(* IEC 61131-3 sources: AXOpen/src/templates.simple/ax/src/templates/starterunit, 8 files *)

(* ---- AutomatSequence.st ---- *)
NAMESPACE axosimple.StarterUnitTemplate
    USING axosimple;
    USING AXOpen.Data;
    USING AXOpen.Core;
    USING System.Strings;

    ///<summary>
    /// Provides automatic mode sequence.
    ///</summary>
    {#ix-set:AttributeName = "<#AUTOMAT#>"}
    {S7.extern=ReadWrite}
    CLASS PUBLIC AutomatSequence
        EXTENDS AXOpen.Core.AxoSequencerContainer IMPLEMENTS IModeContainer
        VAR PUBLIC
            Steps : ARRAY[0..100] OF AxoStep;

            _inspectionResult: BOOL;
            _inspectionValue: LREAL;
            _inspectionData: STRING;

            _comprehensiveResult: AXOpen.Inspectors.AxoComprehensiveResult;
        END_VAR

        VAR PRIVATE
            Objs : REF_TO axosimple.StarterUnitTemplate.UnitObjects;
            Components : REF_TO axosimple.StarterUnitTemplate.Components;
            ProcessDataManager : REF_TO axosimple.StarterUnitTemplate.ProcessDataManager;
            ProcessSettingsManager : REF_TO axosimple.StarterUnitTemplate.FragmentProcessDataManger;
            TechnologySettingsManager : REF_TO axosimple.StarterUnitTemplate.TechnologyDataManager;

            EntityHeader : REF_TO axosimple.EntityData;
            ProcessData : REF_TO axosimple.StarterUnitTemplate.ProcessData;
            ProcessSettings : REF_TO axosimple.StarterUnitTemplate.ProcessData;
            TechnologySettings : REF_TO axosimple.StarterUnitTemplate.TechnologyData;

            _currentId : STRING;

            _dialogAnswer : eDialogAnswer;
            _externalCloseOkSignal : BOOL;
        END_VAR

        METHOD INTERNAL Run
            VAR_INPUT
                _parent : AXOpen.Core.IAxoObject;
                _unitObjects : REF_TO UnitObjects;
            END_VAR

            IF Objs = NULL THEN
                Objs := _unitObjects;

                Components := Objs^.Components;
                ProcessDataManager := Objs^.ProcessData;
                ProcessSettingsManager := Objs^.ProcessSettings;
                TechnologySettingsManager := Objs^.TechnologySettings;

                EntityHeader := REF(ProcessDataManager^.Shared.Entity);
                ProcessData :=  REF(ProcessDataManager^.DataManger.Payload);
                ProcessSettings :=  REF(ProcessSettingsManager^.Payload);
                TechnologySettings :=  REF(TechnologySettingsManager^.DataManger.Payload);

            END_IF;

            SUPER.Run(_parent);
        END_METHOD
        ///<summary>
        /// Contains logic of the steps of this sequence
        ///</summary>

        METHOD OVERRIDE Main
            VAR
                forIterator : INT := 0;
                dialogTimeOut : TIME:= t#3000ms;
            END_VAR

            IF (Components = NULL OR ProcessDataManager = NULL) THEN
                RETURN;
            END_IF;
            // This sequecner executes the steps in cycles from top to bottom
            // in the same order they are written in the program
            // Each step in the sequence must can be used only once.
            // This sets the sequence to run in cycles (top-botton-top and again).
            THIS.SequenceMode := eAxoSequenceMode#Cyclic;

            IF (Steps[0].Execute(THIS, TRUE, '<#GET ID#>')) THEN
                //-------------------------------------------------------
                Objs^._inspectorDialog.Restore();

                // copy data from setting to station data -> it's a problem with override checks identity
                //ProcessData^ :=  ProcessSettings^;

                ProcessData^.PartPresence.Data()^.FailTime := TIME#3s;
                ProcessData^.LoadPosition.Data()^.FailTime := TIME#3s;
                ProcessData^.JigDataMatrixCode.Data()^.FailTime := TIME#3s;

                ProcessData^.PartPresence.Data()^.PassTime := TIME#2.5s;
                ProcessData^.LoadPosition.Data()^.PassTime := TIME#2s;
                ProcessData^.JigDataMatrixCode.Data()^.PassTime := TIME#2s;

                ProcessData^.PartPresence.Data()^.RequiredStatus := TRUE;
                ProcessData^.LoadPosition.Data()^.RequiredMin := 1000.0;
                ProcessData^.LoadPosition.Data()^.RequiredMax := 2000.0;
                ProcessData^.JigDataMatrixCode.Data()^.RequiredStatus := 'passCode';

                _currentId := 'newProducedPart';
                THIS.MoveNext();
                //-------------------------------------------------------
            END_IF;

            IF (Steps[1].Execute(THIS, TRUE, '<#GET DATA#>')) THEN
                //-------------------------------------------------------
                IF (ProcessDataManager^.CreateOrUpdate(_currentId).IsDone()) THEN
                    THIS.MoveNext();
                END_IF;
                //-------------------------------------------------------
            END_IF;

            IF (Steps[2].Execute(THIS, TRUE, '<#Dialog notify#>')) THEN
                //-------------------------------------------------------
                _externalCloseOkSignal := CurrentStep.Duration > dialogTimeOut;

                _dialogAnswer := Objs^._dialog.ShowWithExternalClose(THIS, _externalCloseOkSignal)
                .WithOK()
                .WithType(eDialogType#Info)
                .WithCaption('Info caption!')
                .WithText('Info - dialog will be closed by external timeout 2s!').Answer();

                IF( _dialogAnswer = eDialogAnswer#Ok) THEN
                    THIS.MoveNext();
                END_IF;
                //-------------------------------------------------------
            END_IF;

            IF (Steps[3].Execute(THIS, TRUE, '<#Dialog success#>')) THEN
                //-------------------------------------------------------
                _externalCloseOkSignal := CurrentStep.Duration > dialogTimeOut;

                    _dialogAnswer := Objs^._dialog.ShowWithExternalClose(THIS, _externalCloseOkSignal)
                    .WithOK()
                    .WithType(eDialogType#Success)
                    .WithCaption('Success caption!')
                    .WithText('Success - dialog will be closed by external timeout 2s!').Answer();

                    IF( _dialogAnswer = eDialogAnswer#Ok) THEN
                        THIS.MoveNext();
                    END_IF;
                //-------------------------------------------------------
            END_IF;

            IF (Steps[4].Execute(THIS, TRUE, '<#Dialog Warning#>')) THEN
                //-------------------------------------------------------
                _externalCloseOkSignal := CurrentStep.Duration > dialogTimeOut;

                    _dialogAnswer := Objs^._dialog.ShowWithExternalClose(THIS, _externalCloseOkSignal)
                    .WithYesNo()
                    .WithType(eDialogType#Warning)
                    .WithCaption('Warning caption!')
                    .WithText('Warning - dialog will be closed by external timeout 2s!').Answer();

                    IF( _dialogAnswer = eDialogAnswer#Ok) THEN
                        THIS.MoveNext();
                    END_IF;
                //-------------------------------------------------------
            END_IF;

            IF (Steps[5].Execute(THIS, TRUE, '<#Dialog danger#>')) THEN
                //-------------------------------------------------------
                _externalCloseOkSignal := CurrentStep.Duration > dialogTimeOut;

                    _dialogAnswer := Objs^._dialog.ShowWithExternalClose(THIS, _externalCloseOkSignal)
                    .WithYesNoCancel()
                    .WithType(eDialogType#Warning)
                    .WithCaption('Danger caption!')
                    .WithText('Danger - dialog will be closed by external timeout 2s!').Answer();

                    IF( _dialogAnswer = eDialogAnswer#Ok) THEN
                        THIS.MoveNext();
                    END_IF;
                //-------------------------------------------------------
            END_IF;

            IF (Steps[6].Execute(THIS, TRUE, 'Example Digital inspection')) THEN
                //-------------------------------------------------------
                ProcessData^.PartPresence.WithCoordinator(THIS).Inspect(THIS,_inspectionResult)
                .UpdateComprehensiveResult(_comprehensiveResult)
                .OnFail()
                .CarryOn();
                //-------------------------------------------------------
            END_IF;

            IF (Steps[7].Execute(THIS, TRUE, 'Example Analog inspection')) THEN
                //-------------------------------------------------------
                _inspectionValue := -5500;

                ProcessData^.LoadPosition.WithCoordinator(THIS)
                .Inspect(THIS,_inspectionValue)
                .UpdateComprehensiveResult(_comprehensiveResult)
                .OnFail()
                .Dialog( inRetryStep := Steps[50], inTerminateStep := Steps[60], inoDialog := Objs^._inspectorDialog);
                //-------------------------------------------------------
            END_IF;

            IF (Steps[8].Execute(THIS, TRUE, 'Example Data inspection')) THEN
                //-------------------------------------------------------
                _inspectionData := 'tempCode';

                ProcessData^.JigDataMatrixCode.WithCoordinator(THIS)
                .Inspect(THIS,_inspectionData)
                .UpdateComprehensiveResult(_comprehensiveResult)
                .OnFail()
                .Dialog( inRetryStep := Steps[70], inTerminateStep := Steps[80], inoDialog := Objs^._inspectorDialog);
                //-------------------------------------------------------
            END_IF;

            FOR forIterator := 10 TO 89 BY 1 DO
                IF (Steps[forIterator].Execute(THIS, TRUE,Concat('DO SOMETHING -A-',ToString(forIterator)) )) THEN
                    //-------------------------------------------------------
                    IF CurrentStep.Duration > TIME#50ms THEN
                        THIS.MoveNext();
                    END_IF;
                    //-------------------------------------------------------
                END_IF;
            END_FOR;

            IF (Steps[99].Execute(THIS, TRUE,'<#UPDATE DATA#>')) THEN
                //-------------------------------------------------------
                IF (ProcessDataManager^.Update(_currentId).IsDone()) THEN
                    THIS.MoveNext();
                END_IF;
                //-------------------------------------------------------
            END_IF;

            // This will close the sequence and will return to the first step.
            THIS.Close(Steps[100]);
        END_METHOD
    END_CLASS

END_NAMESPACE

(* ---- Comonents.st ---- *)
NAMESPACE axosimple.StarterUnitTemplate
    USING axosimple;
    USING AXOpen.Data;
    USING AXOpen.Core;
    USING System.Strings;

    ///<summary>
    /// Groups components of this controller unit.
    ///</summary>
    {S7.extern=ReadWrite}
    CLASS Components
        EXTENDS AXOpen.Core.AxoObject
        VAR PUBLIC
            // HERE DECLARE COMPONENTS USED BY THIS CONTROLLED UNIT
            // HorizontalCylinder : AXOpen.Components.Pneumatics.AxoCylinder;
            // VerticalCylinder : AXOpen.Components.Pneumatics.AxoCylinder;
            // GripperCylinder : AXOpen.Components.Pneumatics.AxoCylinder;
            // DMCReader : AXOpen.Components.Cognex.Vision.v_6_0_0_0.AxoDataman;
            // PartPresenceSensor : AXOpen.Elements.AxoDi;
        END_VAR

        METHOD PUBLIC Update
            VAR_INPUT
                parent : IAxoObject;
            END_VAR
            VAR_IN_OUT
                Inputs : axosimple.Inputs;
                Outputs : axosimple.Outputs;
            END_VAR
            THIS.Initialize(parent);
            // HERE INITIALIZE YOUR COMPONENTS
            // HorizontalCylinder.Run(THIS, Inputs.B0[0], Inputs.B0[1], Outputs.B0[0], Outputs.B0[1]);
            // VerticalCylinder.Run(THIS, Inputs.B0[2], Inputs.B0[3], Outputs.B0[2], Outputs.B0[3]);
            // GripperCylinder.Run(THIS, Inputs.B0[4], Inputs.B0[5], Outputs.B0[4], Outputs.B0[5]);
        END_METHOD
    END_CLASS
END_NAMESPACE

(* ---- GroundSequence.st ---- *)
NAMESPACE axosimple.StarterUnitTemplate
    USING axosimple;
    USING AXOpen.Data;
    USING AXOpen.Core;
    USING System.Strings;

    ///<summary>
    /// Provides ground mode sequence.
    ///</summary>
    {#ix-set:AttributeName = "<#GROUND#>"}
    {S7.extern=ReadWrite}
    CLASS PUBLIC GroundSequence
        EXTENDS AXOpen.Core.AxoSequencerContainer
        VAR PUBLIC
            Steps : ARRAY[0..20] OF AxoStep;
            MoveToWork : AxoTask;
        END_VAR
        VAR PRIVATE
            Objs : REF_TO axosimple.StarterUnitTemplate.UnitObjects;
            Components : REF_TO Components;
            ProcessData : REF_TO ProcessDataManager;
            ProcessSettings : REF_TO FragmentProcessDataManger;
            TechnologySettings : REF_TO TechnologyDataManager;
            PersistentSettings : REF_TO AxoDataPersistentExchange;

            _currentId : STRING;
            techSetttingsId : STRING;
        END_VAR

        METHOD INTERNAL Run
            VAR_INPUT
                _parent : IAxoObject;
                _unitObjects : REF_TO axosimple.StarterUnitTemplate.UnitObjects;
            END_VAR

            IF Objs = NULL THEN
                Objs := _unitObjects;

                Components := Ref(Objs^.Components);
                ProcessData := Objs^.ProcessData;
                ProcessSettings := Objs^.ProcessSettings;
                TechnologySettings := Objs^.TechnologySettings;
                PersistentSettings := Objs^.Global^.PersistentData;
            END_IF;

            SUPER.Run(_parent);
        END_METHOD

        ///<summary>
        /// Contains logic of the steps of this sequence
        ///</summary>
        METHOD PROTECTED OVERRIDE Main
            VAR
                taskState :IAxoTaskState;
            END_VAR;
            // IF (Components = NULL OR ProcessData = NULL) THEN
            //     RETURN;
            // END_IF;
            // This sequecner executes the steps in cycles from top to bottom
            // in the same order they are written in the program
            // Each step in the sequence must can be used only once.
            // This sets the sequence to run once (top-botton) and stops with done after closing.
            THIS.SequenceMode := eAxoSequenceMode#RunOnce;

            // This is more verbose but also more versatile way of executing step logic.
            IF (Steps[0].Execute(THIS, TRUE, '<#RESTORE#>')) THEN
                //-------------------------------------------------------
                TechnologySettings^.Restore();
                ProcessSettings^.Restore();
                ProcessData^.Restore();

                THIS.MoveNext();
                //-------------------------------------------------------
            END_IF;

            IF (Steps[1].Execute(THIS, TRUE, '<#READ PERSISTENT SETTINGS#>')) THEN
                //-------------------------------------------------------
                IF CurrentStep.IsFirstEntryToStep() THEN
                    ;// some special initialization
                END_IF;

                CASE TO_INT( THIS.GetMicroStepValue()) OF
                    0 :
                        IF PersistentSettings^.InvokeEntityExist(THIS ,'') THEN
                            THIS.SetMicroStepValue(UINT#10);
                        END_IF;

                    10 :
                        IF PersistentSettings^.IsEntityExistDone(THIS) THEN
                            IF PersistentSettings^.EntityExistResult() THEN
                                THIS.SetMicroStepValue(UINT#40); // default data exist
                            ELSE
                                THIS.SetMicroStepValue(UINT#20); // no data exist
                            END_IF;
                        END_IF;

                    20 :
                        IF PersistentSettings^.InvokeUpdateAll(THIS) THEN // data not exist -> udate all to DB
                            THIS.SetMicroStepValue(UINT#30);
                        END_IF;

                    30:
                        IF PersistentSettings^.IsUpdateAllDone(THIS) THEN
                            THIS.SetMicroStepValue(UINT#40); // all was updated to DB
                        END_IF;

                    40 :
                        IF PersistentSettings^.InvokeRead(THIS, '') THEN // read default group
                            THIS.SetMicroStepValue(UINT#50);
                        END_IF;
                    50 :
                        IF PersistentSettings^.IsReadDone(THIS) THEN
                                THIS.MoveNext(); // just default group was readed
                        END_IF;
                    ELSE
                        THIS.SetMicroStepValue(UINT#0);
                END_CASE;

                //-------------------------------------------------------
            END_IF;

            IF (Steps[5].Execute(THIS, TRUE, '<#READ TECHNOLOGY SETTINS#>')) THEN
                //-------------------------------------------------------
                IF CurrentStep.IsFirstEntryToStep() THEN

                    IF Objs^.Global^.TechnologySettings^.Common.Entity.DataEntityId <> '' THEN
                       techSetttingsId := Objs^.Global^.TechnologySettings^.Common.Entity.DataEntityId; // TAKE GLOGAL TECHNOLOGY SETTINGS ID

                    ELSIF Objs^.TechnologySettings^.Shared.Entity.DataEntityId <> '' THEN // TAKE LAST LOADED FOR STATION
                        techSetttingsId := Objs^.TechnologySettings^.Shared.Entity.DataEntityId;

                    ELSIF Objs^.LastTechnologySettings <> '' THEN // TAKE LAST LOADED FROM PERSISTENT
                        techSetttingsId := Objs^.LastTechnologySettings;
                    ELSE
                        Objs^.LastTechnologySettings := 'default'; // FORCE DEFAULT VALUE
                        techSetttingsId := Objs^.LastTechnologySettings;
                    END_IF;

                    IF Objs^.Global^.TechnologySettings^.Common.Entity.DataEntityId = Objs^.TechnologySettings^.Shared.Entity.DataEntityId then
                        //THIS.MoveNext(); // you can skip loading...
                        ;
                    end_if;

                else
                    IF(TechnologySettings^.Read( techSetttingsId ).IsDone()) THEN
                        THIS.MoveNext();
                    END_IF;
                END_IF;
                //-------------------------------------------------------
            END_IF;

            IF (Steps[6].Execute(THIS, TRUE, '<#DO SOMETHING#>')) THEN
                //-------------------------------------------------------
                IF CurrentStep.Duration > TIME#2s THEN
                    THIS.MoveNext();
                END_IF;
                //-------------------------------------------------------
            END_IF;

            IF (Steps[19].Execute(THIS, TRUE, '<#SAVE DATA#>')) THEN
                //-------------------------------------------------------
                CASE TO_INT( THIS.GetMicroStepValue()) OF
                    0 :
                        IF ProcessData^.Shared.Entity.DataEntityId <> '' THEN
                            _currentId := ProcessData^.Shared.Entity.DataEntityId;
                            THIS.SetMicroStepValue(UINT#10);

                        ELSE // FIST RUN OR WITHOUT DATA
                            THIS.MoveNext();
                        END_IF;

                    10 : // update part as a corrupted a interrupted
                        ProcessData^.Shared.Entity.WasReset := true;
                        IF ProcessData^.Update(_currentId).IsDone() THEN
                                THIS.MoveNext();
                        END_IF;
                    ELSE
                        THIS.SetMicroStepValue(UINT#0);
                END_CASE;
                //-------------------------------------------------------
            END_IF;

            // This will close the sequence and will return to the first step.
            THIS.Close(Steps[20]);
        END_METHOD
    END_CLASS
END_NAMESPACE

(* ---- ProcessData.st ---- *)
NAMESPACE axosimple.StarterUnitTemplate
    USING axosimple;
    USING AXOpen.Data;
    USING AXOpen.Core;
    USING System.Strings;

    {S7.extern=ReadWrite}
    CLASS ProcessData
        EXTENDS AXOpen.Data.AxoDataEntity
        VAR PUBLIC
            CounterDelay : ULINT;
        END_VAR
    END_CLASS
END_NAMESPACE

(* ---- ServiceMode.st ---- *)
NAMESPACE axosimple.StarterUnitTemplate
    USING axosimple;
    USING AXOpen.Data;
    USING AXOpen.Core;
    USING System.Strings;

    ///<summary>
    /// Provides logic for service/manual/maintenance mode.
    ///</summary>
    {#ix-set:AttributeName = "<#SERVICE#>"}
    {S7.extern=ReadWrite}
    CLASS PUBLIC ServiceMode
        EXTENDS AXOpen.Core.AxoTask
        ///<summary>
        /// Runs service mode logic. This method must be called cyclically.
        ///</summary>

        METHOD PUBLIC Run
            VAR_INPUT
                parent : IAxoObject;
            END_VAR
            VAR_IN_OUT
                components : Components;
            END_VAR
            THIS.Initialize(parent);
            IF THIS.Execute() THEN
                THIS.Handle(components);
            END_IF;
        END_METHOD

        METHOD PRIVATE Handle
            VAR_IN_OUT
                components : Components;
            END_VAR
            ;
            // HERE CALL LOGIC FOR MANUAL/SERICE OPERATIONS
            // components.HorizontalCylinder.ActivateManualControl();
            // components.VerticalCylinder.ActivateManualControl();
            // components.GripperCylinder.ActivateManualControl();
        END_METHOD
    END_CLASS
END_NAMESPACE

(* ---- TechnologyData.st ---- *)
NAMESPACE axosimple.StarterUnitTemplate
    USING axosimple;
    USING AXOpen.Data;
    USING AXOpen.Core;
    USING System.Strings;

    CLASS TechnologyData
        EXTENDS AXOpen.Data.AxoDataEntity
        VAR PUBLIC

            Header : axosimple.TechnologyUnitHeader;

            HeatingTemperature   : REAL;

        END_VAR
    END_CLASS
END_NAMESPACE

(* ---- Unit.st ---- *)
NAMESPACE axosimple.StarterUnitTemplate
    USING axosimple;
    USING AXOpen.Data;
    USING AXOpen.Core;
    USING System.Strings;

    ///<summary>
    /// Represents controlled units and high level task coordination.
    ///</summary>
    CLASS Unit
        EXTENDS AXOpen.Core.AxoObject IMPLEMENTS axosimple.IUnit
        VAR PUBLIC
                        ///<summary>
            /// Provide access to unit objets, that are used into sequnces.
            ///</summary>
            UnitObjects  : UnitObjects;

            ///<summary>
            /// Ground sequence. Contains logic that brings the unit into initial state.
            ///</summary>
            GroundSequence : GroundSequence;

            ///<summary>
            /// Automatic sequence. Contains logic for automatic operations of this unit.
            ///</summary>
            AutomatSequence : AutomatSequence;

            ///<summary>
            /// Service mode contains logic for service/manual operations.
            ///</summary>
            ServiceMode : ServiceMode;
        END_VAR
        ///<summary>
        /// Runs this unit.
        ///</summary>

        METHOD PUBLIC Run
            VAR_INPUT
                parent : IAxoContext;
            END_VAR
            VAR_IN_OUT
                ///<summary>
                /// Hardware input structure
                ///</summary>
                Inputs : axosimple.Inputs;
                ///<summary>
                /// Hardware output structure
                ///</summary>
                Outputs : axosimple.Outputs;
            END_VAR
            THIS.Initialize(parent);
            THIS.Execute(Inputs, Outputs);
        END_METHOD

        METHOD PRIVATE Execute
            VAR_IN_OUT
                Inputs : axosimple.Inputs;
                Outputs : axosimple.Outputs;
            END_VAR

            // Component I/O immange and management handling.
             UnitObjects.Components.Update(THIS, Inputs, Outputs);
             // Process data manager
             UnitObjects.ProcessData^.Run(THIS);
             // Technology data manager
             UnitObjects.TechnologySettings^.Run(THIS);
             // Handles ground sequence
             GroundSequence.Run(THIS, REF(UnitObjects));
             // Restores other states when Ground executes
             IF (GroundSequence.IsBusy()) THEN
                 AutomatSequence.Restore();
                 ServiceMode.Restore();
             END_IF;

             // Handles automatic sequence (ground must be previously done)
             AutomatSequence.IsDisabled := GroundSequence.Status <> eAxoTaskState#Done;
             AutomatSequence.Run(THIS, REF(UnitObjects));
             // Handles service/manual mode
             ServiceMode.Run(THIS, UnitObjects.Components);

             IF ServiceMode.IsBusy() THEN
                 GroundSequence.Restore();
                 AutomatSequence.Restore();
             END_IF;

            // remember last selected technolgy identifier
            // if  (UnitObjects.LastTechnologySettings <> '') THEN
            //     IF UnitObjects.LastTechnologySettings <> UnitObjects.TechnologySettings^.DataManger.Payload.DataEntityId THEN

            //        IF UnitObjects.PersistentData^.InvokeUpdate(THIS, '') THEN
            //             UnitObjects.LastTechnologySettings :=  UnitObjects.TechnologySettings^.DataManger.Payload.DataEntityId;
            //        END_IF;
            //     END_IF;
            // END_IF;
        END_METHOD
    END_CLASS

END_NAMESPACE

(* ---- UnitObjects.st ---- *)
NAMESPACE axosimple.StarterUnitTemplate

    USING axosimple;
    USING AXOpen.Data;
    USING AXOpen.Core;
    USING System.Strings;

    {S7.extern=ReadWrite}
    CLASS PUBLIC UnitObjects EXTENDS axosimple.BaseUnit.UnitObjects
        VAR PUBLIC
            ///<summary>
            /// Handles and intializes components used by this unit.
            ///</summary>
            Components : REF_TO axosimple.StarterUnitTemplate.Components;

            ///<summary>
            /// Provides access to process data manager of this unit
            ///</summary>
            ProcessSettings : REF_TO axosimple.StarterUnitTemplate.FragmentProcessDataManger;

            ///<summary>
            /// Provides access to process data manager of this unit
            ///</summary>
            ProcessData : REF_TO axosimple.StarterUnitTemplate.ProcessDataManager;

            ///<summary>
            /// Provides access to process data manager of this unit
            ///</summary>
            TechnologySettings : REF_TO axosimple.StarterUnitTemplate.TechnologyDataManager;

            {#ix-attr:[AXOpen.Data.PersistentAttribute("StarterUnitTemplate")]}
            SpecialSettings :STRING[64] ;

            // https://ix-ax.github.io/AXOpen/core/docs/AXODIALOG.html#closing-a-dialog-with-external-signal
            _dialog : AXOpen.Core.AxoDialog;

            // https://ix-ax.github.io/AXOpen/core/docs/AXOALERTDIALOG.html#invoking-alerts-from-plc
            _alertDialog : AXOpen.Core.AxoAlertDialog;

            // it needs to be handle from auto or ground sequnce
            _inspectorDialog       : AXOpen.Inspectors.AxoInspectorDialog;

        END_VAR
    END_CLASS

END_NAMESPACE
